SUBAPPLICATION Uebung_012d_AX (* Numeric Value Input PHYS und Speichern NVS *)
  (* Standard: 61499-2; Description: Copyright (c) 2026 Meisterschulen am Ostbahnhof This program and the accompanying materials are made available under the terms of the Eclipse Public License 2.0 which is available at https://www.eclipse.org/legal/epl-2.0/ SPDX-License-Identifier: EPL-2.0 *)
  (* Version 1.0, 2026-04-24, Franz Höpfinger, Meisterschulen am Ostbahnhof, AR adapter variant of Uebung_012d *)
  PACKAGE Uebungen;
  IMPORT Uebungen::const::NVS::NVS_Keys::KEY_I1_STORE;
  IMPORT Uebungen::const::UT::DefaultPool_Numeric::InputNumber_I3_N;
  IMPORT Uebungen::const::UT::DefaultPool_Numeric::OutputNumber_N3_N;
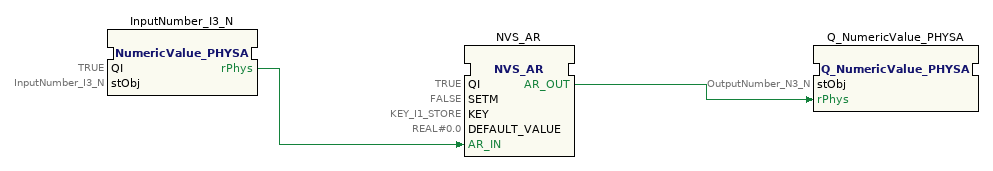
  FBS
    InputNumber_I3_N : isobus::UT::io::NumericValue::NumericValue_PHYSA(QI := TRUE, stObj := InputNumber_I3_N);
    NVS_AR : logiBUS::storage::esp32_nvs::NVS_AR(QI := TRUE, SETM := FALSE, KEY := KEY_I1_STORE, DEFAULT_VALUE := REAL#0.0);
    Q_NumericValue_PHYSA : isobus::UT::Q::Q_NumericValue_PHYSA(stObj := OutputNumber_N3_N);
  END_FBS
  ADAPTER_CONNECTIONS
    NVS_AR.AR_OUT TO Q_NumericValue_PHYSA.rPhys;
    InputNumber_I3_N.rPhys TO NVS_AR.AR_IN;
  END_CONNECTIONS
END_SUBAPPLICATION
